Staubli VAL3: TubePoint.pgx

public program TubePoint(trsf& x_trSource[], num x_nAngle, trsf& x_trDest[], bool& x_bRes)
  local num l_ni
  local frame l_fFrame
  local num l_Dia
  local point l_pBuff
  local trsf l_trSupport
  local trsf l_trBuff[3]
begin
 //切管子应用
 //设置三点和一个角度就可以进行实现

  call Circumcircle(x_trSource,l_trSupport,l_Dia,x_bRes)
  if !x_bRes
    return
  endIf
  call CirClePoint(l_trSupport,l_Dia,x_trDest,x_bRes)
  if !x_bRes
    return
  endIf
  x_trDest[20]=l_trSupport




  //对点在对应坐标系下进行偏移
  for l_ni=0 to 3
    l_trBuff[0]=x_trDest[l_ni]
    l_trBuff[1]=l_trSupport
    l_trBuff[2]=x_trDest[l_ni+1]
    call SetFrame(l_trBuff,l_fFrame,x_bRes)
    if !x_bRes
      return
    endIf
    l_pBuff.trsf=x_trDest[l_ni]
    link(l_pBuff,world)
   l_pBuff=compose(l_pBuff,l_fFrame,{0,0,0,0,-x_nAngle,0})
    x_trDest[l_ni]=position(l_pBuff,world)
  endFor
  x_trDest[4]=x_trDest[0]


end
